// TIA Portal V17 export
// export: Created 2025-03-10T13:12:16.5070959Z, ExportSetting WithDefaults, DisplayName Totally Integrated Automation Portal, DisplayVersion V17 Update 8, DisplayName TIA Portal Openness, DisplayVersion V17 Update 8, DisplayName TIA Portal Version Control Interface, DisplayVersion V17, DisplayName SINAMICS Startdrive Advanced, DisplayVersion V17 SP2, DisplayName SINAMICS Startdrive G110M, G120, G120C, G120D, G120P, G115D, DisplayVersion V17 SP2, DisplayName SINAMICS Startdrive G130, G150, S120, S150, SINAMICS MV, S210, DisplayVersion V17 SP2, DisplayName STEP 7 Professional, DisplayVersion V17 Update 8, DisplayName SINUMERIK ONE STEP 7 Toolbox, DisplayVersion V17 Update 12, DisplayName SINUMERIK 840D sl STEP 7 Toolbox, DisplayVersion V17 Update 12, DisplayName STEP 7 Safety, DisplayVersion V17 Update 6, DisplayName WinCC Advanced, DisplayVersion V17 Update 8
TYPE "LOAD_UNLOAD_ETXETAR_ROBOT_CELL"
// stored: IsFailsafeCompliant false
   STRUCT
      FROM_ROBOT_CELL : Struct
         PART_A_LOADED : Bool;   // PART 1 LOADED ARM 1 / PART A LOADED 1
         PART_A_UNLOADED : Bool;   // PART 1 UNLOADED ARM 1 / PART A UNLOADED 1
         PART_A_LOADED_P : Bool;   // PART 1 LOADED ARM 1 PULSE / PART A LOADED 1 PULSE
         PART_A_UNLOADED_P : Bool;   // PART 1 UNLOADED ARM 1 PULSE / PART A UNLOADED 1 PULSE
      END_STRUCT;
      TO_ROBOT_CELL : Struct
         REQ_LOAD_PART_A : Bool;   // REQUEST LOAD PART 1 ARM 1 / REQUEST LOAD PART A-1
         REQ_UNLOAD_PART_A : Bool;   // REQUEST UNLOAD PART 1 ARM 1 / REQUEST UNLOAD PART A-1
      END_STRUCT;
   END_STRUCT;
END_TYPE
